(* IEC 61131-3 sources: AXOpen/src/components.elements/app/src/Documentation, 1 file *)

(* ---- DocumentationContext.st ---- *)
USING AXOpen.Core;

NAMESPACE AXOpen.Components.Elements
    {S7.extern=ReadWrite}
    CLASS DocumentationContext EXTENDS AXOpen.Core.AxoContext
        VAR PUBLIC
            Cu : DocumentationControllUnit;
        END_VAR
        VAR
            _rootObject : AxoObject;
        END_VAR
        METHOD PROTECTED OVERRIDE Main
            THIS.InitializeRootObject(_rootObject);
            Cu.Main(_rootObject);
        END_METHOD
    END_CLASS

    {S7.extern=ReadWrite}
    CLASS DocumentationControllUnit EXTENDS AXOpen.Core.AxoObject

        //<AxoDiDeclaration>
        VAR PUBLIC
            _testDi : AXOpen.Components.Elements.AxoDi;
        END_VAR
        //</AxoDiDeclaration>

        //<AxoDiInitializationArgumentsDeclaration>
        VAR PUBLIC
            _testsignal : BOOL;
        END_VAR
        //</AxoDiInitializationArgumentsDeclaration>

        //<AxoDoDeclaration>
        VAR PUBLIC
            _testDo : AXOpen.Components.Elements.AxoDo;
        END_VAR
        //</AxoDoDeclaration>

        //<AxoDoInitializationArgumentsDeclaration>
        VAR PUBLIC
            _testInOutSignal : BOOL;
        END_VAR
        //</AxoDoInitializationArgumentsDeclaration>

        //<AxoAiDeclaration>
        VAR PUBLIC
            _testAi : AXOpen.Components.Elements.AxoAi;
        END_VAR
        //</AxoAiDeclaration>

        //<AxoAiInitializationArgumentsDeclaration>
        VAR PUBLIC
            _testAiInput : DINT := DINT#10;
        END_VAR
        //</AxoAiInitializationArgumentsDeclaration>

        //<AxoAoDeclaration>
        VAR PUBLIC
            _testAo : AXOpen.Components.Elements.AxoAo;
        END_VAR
        //</AxoAoDeclaration>

        //<AxoAoInitializationArgumentsDeclaration>
        VAR PUBLIC
            _testAoOutput : DINT;
        END_VAR
        //</AxoAoInitializationArgumentsDeclaration>

        //<AxoCarouselDeclaration>
        VAR PUBLIC
            _testCarousel : AXOpen.Components.Elements.AxoRotaryIndexingTable;
        END_VAR
        //</AxoCarouselDeclaration>

        //<AxoCarouselInitializationArgumentsDeclaration>
        VAR PUBLIC
                _testCarouselSafetyCondition    :   BOOL;
            	_testCarouselInPosition         :   BOOL;
            	_testCarouselInPrecisePosition  :   BOOL;
                _testCarouselCodingPosition     :   UINT;
                _testCarouselEnableTurn         :   BOOL;
                _testCarouselStartTurn          :   BOOL;

                _testCarouselSuspend1           :   BOOL;
                _testCarouselSuspend2           :   BOOL;
                _testCarouselSuspend3           :   BOOL;
            END_VAR
        //</AxoCarouselInitializationArgumentsDeclaration>

        METHOD PUBLIC Main
            VAR_INPUT
                inParent  : IAxoObject;
            END_VAR

            SUPER.Run(inParent);

            //<AxoDiManualControl>
            _testDi.ActivateManualControl();
            //</AxoDiManualControl>

            //<AxoDiInitialization>
            _testDi.Run(THIS, _testsignal);
            //</AxoDiInitialization>

            //<AxoDiUsage>
            IF _testDi.IsTrue() THEN
                ;// handle signal on
            END_IF;
            //</AxoDiUsage>

            //<AxoDoManualControl>
            _testDo.ActivateManualControl();
            //</AxoDoManualControl>

            //<AxoDoInitialization>
            _testDo.Run(THIS, _testInOutSignal);
            //</AxoDoInitialization>

            //<AxoDoUsage>
            _testDo.Set();
            //</AxoDoUsage>

            //<AxoAiManualControl>
            _testAi.ActivateManualControl();
            //</AxoAiManualControl>

            //<AxoAiInitialization>
            _testAi.Run(THIS, _testAiInput);
            //</AxoAiInitialization>

            //<AxoAoManualControl>
            _testAo.ActivateManualControl();
            //</AxoAoManualControl>

            //<AxoAoInitialization>
            _testAo.Run(THIS, _testAoOutput);
            //</AxoAoInitialization>

            //<AxoCarouselManualControl>
            _testCarousel.ActivateManualControl();
            //</AxoCarouselManualControl>

            //<AxoCarouselInitialization>
            _testCarousel.Config.ErrorTime:=T#100S;
            _testCarousel.Config.InfoTime:=T#20S;
            _testCarousel.Config.TaskTimeout:=T#200S;
            _testCarousel.Config.Direction:=eAxoRotaryIndexingTableDirection#Cw;
            _testCarousel.Config.NumberOfPositions:=UINT#8;
            _testCarousel.Config.Offset:=UINT#2;

            _testCarousel.Run(  inParent            :=  THIS,
                                inSafetyCondition   :=  _testCarouselSafetyCondition,
                                inPosition          :=  _testCarouselInPosition,
                                inPrecisePosition   :=  _testCarouselInPrecisePosition,
                                inCodingPosition    :=  _testCarouselCodingPosition,
                                outEnableTurn       =>  _testCarouselEnableTurn,
                                outStartTurn        =>  _testCarouselStartTurn);

            _testCarousel.SuspendMovementWhile(_testCarouselSuspend1,'Movement blocked by signal _testCarouselSuspend1');
            _testCarousel.SuspendMovementWhile(_testCarouselSuspend2,'Movement blocked by signal _testCarouselSuspend2');
            _testCarousel.SuspendMovementWhile(_testCarouselSuspend3,'Movement blocked by signal _testCarouselSuspend3');

            //</AxoCarouselInitialization>
        END_METHOD
    END_CLASS
END_NAMESPACE
